// TIA Portal V19 export
TYPE "lexchangetray_typeUnEmn_signalTM_Simulation"
// Type: Bool
// stored: Access Published
   STRUCT
      w : Bool;   // Manual mode parameters for axis control interface
   END_STRUCT;
END_TYPE
